RoboDK station: Name Engraving Scara Robotr.rdk

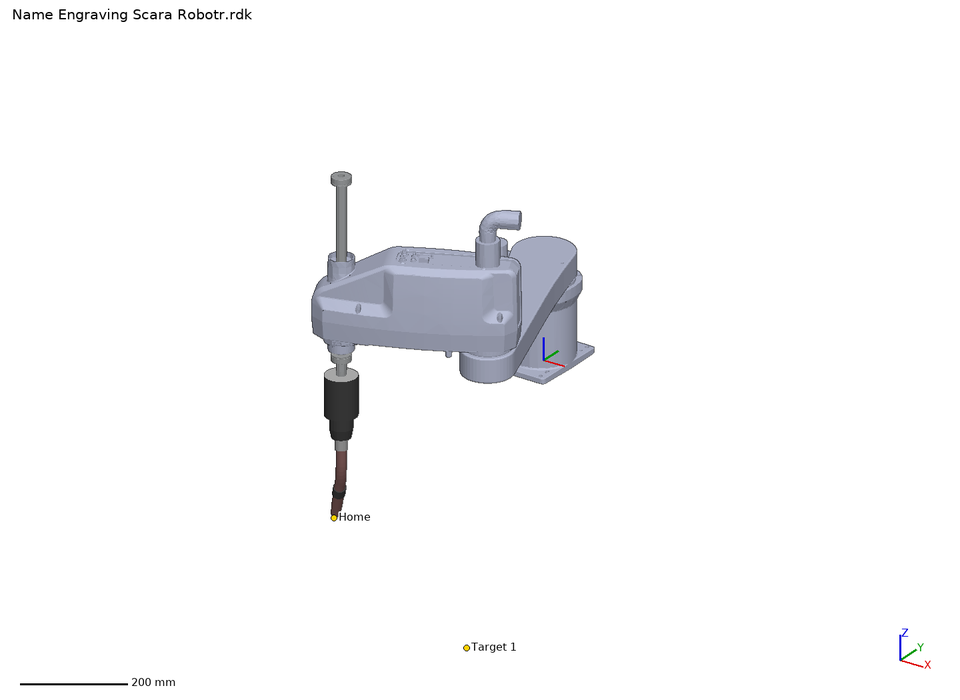
[picture v0: the station drawn from its stored meshes, robots at their saved joint values, targets as dots, program paths as lines]
Station Name Engraving Scara Robotr (saved by RoboDK 5.3.0). Poses are relative to the parent item; angles as X-Y-Z fixed-axis rotations.
  - frame Mitsubishi RH-6CH70 Base at (0, 160.3, 0) mm
    - robot Mitsubishi RH-6CH70: 4 axes, payload 6 kg, reach 700 mm, repeatability 0.025 mm, weight 18 kg
        modified DH rows (alpha deg, a mm, theta deg, d mm): 0, 0, 0, 0; 0, 425, 0, 0; 0, 275, 0, -50 linear; 180, 0, 0, 0
        joint limits [-132, -150, 0, -360] to [132, 150, 200, 360]; home [0, 0, 200, 0]; saved at [-69.237, -84.97, 200, 107.177]
      - tool Welding Gun, TCP at (-91, 0, -340) mm, size 122.1 x 64 x 340.8 mm
    - target Home (Cartesian target) at (-158.96, -450.47, -190) mm, rotated rx 0 ry 0 rz -47.03 deg; joints [-69.237, -84.97, 200, 107.177] of Mitsubishi RH-6CH70
    - target Target 1 (Cartesian target) at (143.61, -455.62, -370.95) mm, rotated rx 0 ry 0 rz -10.11 deg; joints [-32.31, -84.96, 19.05, 107.16] of Mitsubishi RH-6CH70
  - Python program Prog1 (listed below)

--- Python program Prog1 ---
# Draw a hexagon around Target 1
from robolink import *    # RoboDK's API
from robodk import *      # Math toolbox for robots

# Start the RoboDK API:
RDK = Robolink()

# Get the robot (first robot found):
robot = RDK.Item('', ITEM_TYPE_ROBOT)

# Get the reference target by name:
target = RDK.Item('Target 1')
target_pose = target.Pose()
xyz_ref = target_pose.Pos()

# Move the robot to the reference point:
robot.MoveJ(target)

# Draw a hexagon around the reference target:
for i in range(7):
    ang = i*2*pi/6 # Angle = 0,60,120,...,360
    R = 50        # Polygon radius

    # Calculate the new position:
    x = xyz_ref[0] + R*cos(ang) # new X coordinate
    y = xyz_ref[1] + R*sin(ang) # new Y coordinate
    z = xyz_ref[2]              # new Z coordinate
    target_pose.setPos([x,y,z])

    # Move to the new target:
    robot.MoveL(target_pose)

# Trigger a program call at the end of the movement
robot.RunInstruction('Program_Done')

# Move back to the reference target:
robot.MoveL(target)
